(* PLC project SafeLOGIC, BrAutomation SafeDESIGNER  5.24.1.0 *)
(* stored: companyURL http://www.br-automation.com, creationDateTime Tue Aug 26 16:37:49 2025 *)

PROGRAM ELAPSED_TIME_TP

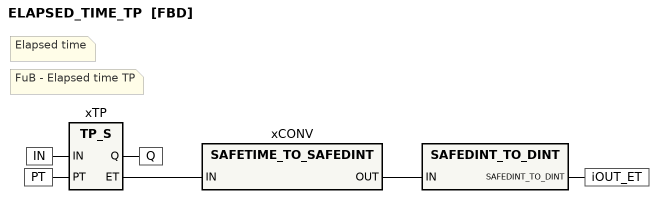
(* FBD diagram, written out as Structured Text *)
(* FuB - Elapsed time TP *)
(* Elapsed time *)
xTP(IN := IN, PT := PT);
Q := xTP.Q;
xCONV(IN := xTP.ET);
iOUT_ET := SAFEDINT_TO_DINT(xCONV.OUT);
END_PROGRAM
